FUNCTION_BLOCK IndexMover EXTENDS FB_Mover
VAR_INPUT
	XtsTrack : IXtsTrack;
	StateMachine : IPmlStateMachine;
END_VAR
VAR_OUTPUT
END_VAR
VAR
	moverSequence : IndexMoverSequence;
	bInit: bool;
END_VAR
VAR_IN_OUT
	StationArray : ARRAY[*] OF IProcess;
END_VAR

IF NOT bInit THEN
	bInit := TRUE;
	_trackLength := XtsTrack.TrackLength;
END_IF
SUPER^();

moverSequence(ThisMover	 := THIS^, 
				XtsTrack := XtsTrack, 
				StateMachine := StateMachine,
				StationArray := StationArray);

END_FUNCTION_BLOCK

(* stored: Version 1.1.0.1, ProductVersion 3.1.4024.11
   POU IndexMover: Id {ae40fee3-92e9-44c7-98fa-7602be1fb9dc}, SpecialFunc None *)
